FUNCTION_BLOCK FB_Sum_Test EXTENDS TcUnit.FB_TestSuite
VAR_INPUT
END_VAR
VAR_OUTPUT
END_VAR
VAR
END_VAR

TwoPlusTwoEqualsFour();
ZeroPlusZeroEqualsZero();

METHOD TwoPlusTwoEqualsFour
VAR
    Sum : FB_Sum;
    Result : UINT;
    ExpectedSum : UINT := 4;
	
	ExpectedProp : BOOL;
	ActualProp: BOOL;
END_VAR
TEST('TwoPlusTwoEqualsFour');
 
Sum(one := 2, two := 2, result => Result);
 
AssertEquals(Expected := ExpectedSum,
             Actual := Result,
             Message := 'The calculation is not correct');
			 
ActualProp := Sum.Prop;
AssertEquals(Expected := ExpectedProp,
             Actual := ActualProp,
             Message := 'Testing prop');			 
 
TEST_FINISHED();
END_METHOD

METHOD ZeroPlusZeroEqualsZero
VAR
    Sum : FB_Sum;
    Result : UINT;
    ExpectedSum : UINT := 0;
END_VAR
TEST('ZeroPlusZeroEqualsZero');
 
Sum(one := 0, two := 0, result => Result);
 
AssertEquals(Expected := ExpectedSum,
             Actual := Result,
             Message := 'The calculation is not correct');
 
TEST_FINISHED();
END_METHOD

END_FUNCTION_BLOCK

(* stored: Version 1.1.0.1, ProductVersion 3.1.4024.12
   POU FB_Sum_Test: Id {abfc6be1-3baf-4283-9266-181748260e6f}, SpecialFunc None
   Method TwoPlusTwoEqualsFour: Id {97cf3e48-0ba0-43da-b044-2ce83d5a63c9}
   Method ZeroPlusZeroEqualsZero: Id {a7c1abba-d08b-4929-8a5e-1574e59bd6bd} *)
